TYPE CM_Sensor_ALM :
STRUCT
END_STRUCT
END_TYPE

(* stored: Version 1.1.0.1, ProductVersion 3.1.4024.12
   DUT CM_Sensor_ALM: Id {348f415d-68a6-42ea-a3cc-7dcfe7b2e044} *)
